{attribute 'no_explicit_call':= 'do not call this POU directly'}
FUNCTION_BLOCK TValueMonitorEx
VAR
    _Changed : BOOL;
    StoredValue : ARRAY[0..7] OF BYTE;
END_VAR

PROPERTY Changed : BOOL
GET
Changed := _Changed;
END_GET
END_PROPERTY

METHOD Reset
VAR_INPUT
END_VAR
MEMSET(
    destAddr := ADR(StoredValue),
    fillByte  := 16#00,
    n        := SIZEOF(StoredValue));
END_METHOD

METHOD Test : BOOL;
VAR_INPUT
    Value : ANY;
END_VAR
_Changed := 0 <>  MEMCMP(
                    pBuf1 := Value.pValue,
                    pBuf2 := ADR(StoredValue),
                    n     := DINT_TO_UDINT(Value.diSize));
    
IF _Changed THEN
    MEMCPY(
        destAddr := ADR(StoredValue),
        srcAddr  := Value.pValue,
        n        := DINT_TO_UDINT(Value.diSize));
END_IF

Test := _Changed;
END_METHOD

END_FUNCTION_BLOCK

(* stored: Version 1.1.0.1, ProductVersion 3.1.4024.3
   POU TValueMonitorEx: Id {cff9be8d-4050-0eea-3e11-96712a333e4f}, SpecialFunc None
   Property Changed: Id {24dee7e2-ee33-09de-271a-026ccd3ad21d}
   Get Get: Id {eca42497-7a64-0abe-1e10-bb9e9e976d8f}
   Method Reset: Id {7e4f45fa-9529-006c-3d68-fc62b1effa1b}
   Method Test: Id {518fc9eb-8ddb-06b9-2161-ed351bdf8745} *)
